# EPICS substitutions: epicsApp/K18MonitorApp/Db/CAENHV1-2.substitutions
file "db/CAENHV_A.template" {

   {crate=1, slot=2, BoardType=SY2527, IP=192.168.30.10, ChMax=24}
}
file "db/CAENHV_B.template" {
   { crate=1, slot=2, name=CH0:V0Set,   ch=1   }
   { crate=1, slot=2, name=CH0:I0Set,   ch=2   }
   { crate=1, slot=2, name=CH0:VMon,    ch=3   }
   { crate=1, slot=2, name=CH0:IMon,    ch=4   }
   { crate=1, slot=2, name=CH0:Pw,      ch=5   }
   { crate=1, slot=2, name=CH0:Status,  ch=6   }
   { crate=1, slot=2, name=CH1:V0Set,   ch=7   }
   { crate=1, slot=2, name=CH1:I0Set,   ch=8   }
   { crate=1, slot=2, name=CH1:VMon,    ch=9   }
   { crate=1, slot=2, name=CH1:IMon,    ch=10  }
   { crate=1, slot=2, name=CH1:Pw,      ch=11  }
   { crate=1, slot=2, name=CH1:Status,  ch=12  }
   { crate=1, slot=2, name=CH2:V0Set,   ch=13  }
   { crate=1, slot=2, name=CH2:I0Set,   ch=14  }
   { crate=1, slot=2, name=CH2:VMon,    ch=15  }
   { crate=1, slot=2, name=CH2:IMon,    ch=16  }
   { crate=1, slot=2, name=CH2:Pw,      ch=17  }
   { crate=1, slot=2, name=CH2:Status,  ch=18  }
   { crate=1, slot=2, name=CH3:V0Set,   ch=19  }
   { crate=1, slot=2, name=CH3:I0Set,   ch=20  }
   { crate=1, slot=2, name=CH3:VMon,    ch=21  }
   { crate=1, slot=2, name=CH3:IMon,    ch=22  }
   { crate=1, slot=2, name=CH3:Pw,      ch=23  }
   { crate=1, slot=2, name=CH3:Status,  ch=24  }
   { crate=1, slot=2, name=CH4:V0Set,   ch=25  }
   { crate=1, slot=2, name=CH4:I0Set,   ch=26  }
   { crate=1, slot=2, name=CH4:VMon,    ch=27  }
   { crate=1, slot=2, name=CH4:IMon,    ch=28  }
   { crate=1, slot=2, name=CH4:Pw,      ch=29  }
   { crate=1, slot=2, name=CH4:Status,  ch=30  }
   { crate=1, slot=2, name=CH5:V0Set,   ch=31  }
   { crate=1, slot=2, name=CH5:I0Set,   ch=32  }
   { crate=1, slot=2, name=CH5:VMon,    ch=33  }
   { crate=1, slot=2, name=CH5:IMon,    ch=34  }
   { crate=1, slot=2, name=CH5:Pw,      ch=35  }
   { crate=1, slot=2, name=CH5:Status,  ch=36  }
   { crate=1, slot=2, name=CH6:V0Set,   ch=37  }
   { crate=1, slot=2, name=CH6:I0Set,   ch=38  }
   { crate=1, slot=2, name=CH6:VMon,    ch=39  }
   { crate=1, slot=2, name=CH6:IMon,    ch=40  }
   { crate=1, slot=2, name=CH6:Pw,      ch=41  }
   { crate=1, slot=2, name=CH6:Status,  ch=42  }
   { crate=1, slot=2, name=CH7:V0Set,   ch=43  }
   { crate=1, slot=2, name=CH7:I0Set,   ch=44  }
   { crate=1, slot=2, name=CH7:VMon,    ch=45  }
   { crate=1, slot=2, name=CH7:IMon,    ch=46  }
   { crate=1, slot=2, name=CH7:Pw,      ch=47  }
   { crate=1, slot=2, name=CH7:Status,  ch=48  }
   { crate=1, slot=2, name=CH8:V0Set,   ch=49  }
   { crate=1, slot=2, name=CH8:I0Set,   ch=50  }
   { crate=1, slot=2, name=CH8:VMon,    ch=51  }
   { crate=1, slot=2, name=CH8:IMon,    ch=52  }
   { crate=1, slot=2, name=CH8:Pw,      ch=53  }
   { crate=1, slot=2, name=CH8:Status,  ch=54  }
   { crate=1, slot=2, name=CH9:V0Set,   ch=55  }
   { crate=1, slot=2, name=CH9:I0Set,   ch=56  }
   { crate=1, slot=2, name=CH9:VMon,    ch=57  }
   { crate=1, slot=2, name=CH9:IMon,    ch=58  }
   { crate=1, slot=2, name=CH9:Pw,      ch=59  }
   { crate=1, slot=2, name=CH9:Status,  ch=60  }
   { crate=1, slot=2, name=CH10:V0Set,  ch=61  }
   { crate=1, slot=2, name=CH10:I0Set,  ch=62  }
   { crate=1, slot=2, name=CH10:VMon,   ch=63  }
   { crate=1, slot=2, name=CH10:IMon,   ch=64  }
   { crate=1, slot=2, name=CH10:Pw,     ch=65  }
   { crate=1, slot=2, name=CH10:Status, ch=66  }
   { crate=1, slot=2, name=CH11:V0Set,  ch=67  }
   { crate=1, slot=2, name=CH11:I0Set,  ch=68  }
   { crate=1, slot=2, name=CH11:VMon,   ch=69  }
   { crate=1, slot=2, name=CH11:IMon,   ch=70  }
   { crate=1, slot=2, name=CH11:Pw,     ch=71  }
   { crate=1, slot=2, name=CH11:Status, ch=72  }
   { crate=1, slot=2, name=CH12:V0Set,  ch=73  }
   { crate=1, slot=2, name=CH12:I0Set,  ch=74  }
   { crate=1, slot=2, name=CH12:VMon,   ch=75  }
   { crate=1, slot=2, name=CH12:IMon,   ch=76  }
   { crate=1, slot=2, name=CH12:Pw,     ch=77  }
   { crate=1, slot=2, name=CH12:Status, ch=78  }
   { crate=1, slot=2, name=CH13:V0Set,  ch=79  }
   { crate=1, slot=2, name=CH13:I0Set,  ch=80  }
   { crate=1, slot=2, name=CH13:VMon,   ch=81  }
   { crate=1, slot=2, name=CH13:IMon,   ch=82  }
   { crate=1, slot=2, name=CH13:Pw,     ch=83  }
   { crate=1, slot=2, name=CH13:Status, ch=84  }
   { crate=1, slot=2, name=CH14:V0Set,  ch=85  }
   { crate=1, slot=2, name=CH14:I0Set,  ch=86  }
   { crate=1, slot=2, name=CH14:VMon,   ch=87  }
   { crate=1, slot=2, name=CH14:IMon,   ch=88  }
   { crate=1, slot=2, name=CH14:Pw,     ch=89  }
   { crate=1, slot=2, name=CH14:Status, ch=90  }
   { crate=1, slot=2, name=CH15:V0Set,  ch=91  }
   { crate=1, slot=2, name=CH15:I0Set,  ch=92  }
   { crate=1, slot=2, name=CH15:VMon,   ch=93  }
   { crate=1, slot=2, name=CH15:IMon,   ch=94  }
   { crate=1, slot=2, name=CH15:Pw,     ch=95  }
   { crate=1, slot=2, name=CH15:Status, ch=96  }
   { crate=1, slot=2, name=CH16:V0Set,  ch=97  }
   { crate=1, slot=2, name=CH16:I0Set,  ch=98  }
   { crate=1, slot=2, name=CH16:VMon,   ch=99  }
   { crate=1, slot=2, name=CH16:IMon,   ch=100 }
   { crate=1, slot=2, name=CH16:Pw,     ch=101 }
   { crate=1, slot=2, name=CH16:Status, ch=102 }
   { crate=1, slot=2, name=CH17:V0Set,  ch=103 }
   { crate=1, slot=2, name=CH17:I0Set,  ch=104 }
   { crate=1, slot=2, name=CH17:VMon,   ch=105 }
   { crate=1, slot=2, name=CH17:IMon,   ch=106 }
   { crate=1, slot=2, name=CH17:Pw,     ch=107 }
   { crate=1, slot=2, name=CH17:Status, ch=108 }
   { crate=1, slot=2, name=CH18:V0Set,  ch=109 }
   { crate=1, slot=2, name=CH18:I0Set,  ch=110 }
   { crate=1, slot=2, name=CH18:VMon,   ch=111 }
   { crate=1, slot=2, name=CH18:IMon,   ch=112 }
   { crate=1, slot=2, name=CH18:Pw,     ch=113 }
   { crate=1, slot=2, name=CH18:Status, ch=114 }
   { crate=1, slot=2, name=CH19:V0Set,  ch=115 }
   { crate=1, slot=2, name=CH19:I0Set,  ch=116 }
   { crate=1, slot=2, name=CH19:VMon,   ch=117 }
   { crate=1, slot=2, name=CH19:IMon,   ch=118 }
   { crate=1, slot=2, name=CH19:Pw,     ch=119 }
   { crate=1, slot=2, name=CH19:Status, ch=120 }
   { crate=1, slot=2, name=CH20:V0Set,  ch=121 }
   { crate=1, slot=2, name=CH20:I0Set,  ch=122 }
   { crate=1, slot=2, name=CH20:VMon,   ch=123 }
   { crate=1, slot=2, name=CH20:IMon,   ch=124 }
   { crate=1, slot=2, name=CH20:Pw,     ch=125 }
   { crate=1, slot=2, name=CH20:Status, ch=126 }
   { crate=1, slot=2, name=CH21:V0Set,  ch=127 }
   { crate=1, slot=2, name=CH21:I0Set,  ch=128 }
   { crate=1, slot=2, name=CH21:VMon,   ch=129 }
   { crate=1, slot=2, name=CH21:IMon,   ch=130 }
   { crate=1, slot=2, name=CH21:Pw,     ch=131 }
   { crate=1, slot=2, name=CH21:Status, ch=132 }
   { crate=1, slot=2, name=CH22:V0Set,  ch=133 }
   { crate=1, slot=2, name=CH22:I0Set,  ch=134 }
   { crate=1, slot=2, name=CH22:VMon,   ch=135 }
   { crate=1, slot=2, name=CH22:IMon,   ch=136 }
   { crate=1, slot=2, name=CH22:Pw,     ch=137 }
   { crate=1, slot=2, name=CH22:Status, ch=138 }
   { crate=1, slot=2, name=CH23:V0Set,  ch=139 }
   { crate=1, slot=2, name=CH23:I0Set,  ch=140 }
   { crate=1, slot=2, name=CH23:VMon,   ch=141 }
   { crate=1, slot=2, name=CH23:IMon,   ch=142 }
   { crate=1, slot=2, name=CH23:Pw,     ch=143 }
   { crate=1, slot=2, name=CH23:Status, ch=144 }
}
